// Converts all alphabetic characters in a string lowercase characters
FUNCTION F_TOLOWER
VAR_INPUT
	sValue : REFERENCE TO STRING; // String of any size
END_VAR
VAR
	i : T_Size;
END_VAR

WHILE sValue[i] <> 0 DO 
	IF sValue[i] >= 65 AND sValue[i]<= 90 THEN sValue[i] := sValue[i] + 32; END_IF
	i := i + 1;
	END_WHILE

END_FUNCTION

(* stored: Version 1.1.0.1, ProductVersion 3.1.4024.4
   POU F_TOLOWER: Id {07aba59d-b3f8-4be4-952e-ac58e1ad8f3c}, SpecialFunc None *)
